{attribute 'GeneratedUsingTerminal: EK1122-0000-0018'}
{attribute addProperty BoxType "EK1122-0000-0018"}
{attribute addProperty Id "Beckhoff_EL72xxsub_EK1100EK1100_AB5A94672"}
{attribute addProperty CRC "1222471656"}
{attribute addProperty Size "2"}
TYPE Beckhoff_EL72xxEK1122_48DD6FE8 EXTENDS EK1122_AB5A9467 :
STRUCT
	{attribute addProperty Name "Beckhoff_EL72xxsub_EK1100"}
	Beckhoff_EL72xxsub_EK1100 : EK1100_AB5A9467;
END_STRUCT
END_TYPE

(* stored: Version 1.2.0.0, ProductVersion 3.1.4024.9
   DUT Beckhoff_EL72xxEK1122_48DD6FE8: Id {759ff562-8070-47d5-8440-1398d0b09a56} *)
